Staubli VAL3: MainKey.pgx

program MainKey(num x_nKey)
  local num l_nKey
begin
  //
  switch x_nKey
    //编辑
    case 271,270
      call OnF1()
    break
    //取反
    case 272
      call OnF2()
    break
    //删除
    case 273
      call OnF3()
    break
    //模拟
    case 274
      call OnF4()
    break
    //
    case 275
    break
    //
    case 276
      call OnF6()
    break
    //save
    case 277
      call OnF7()
    break
    //返回
    case 278,255
      call OnF8("是否返回")
    break
  endSwitch
end
